TYPE ST_ECB :
STRUCT
	Status AT %I* : BOOL;
	Reset AT %Q* : BOOL;
	Name : STRING;
	Description : STRING;
END_STRUCT
END_TYPE

(* stored: Version 1.1.0.1, ProductVersion 3.1.4026.18
   DUT ST_ECB: Id {42e0f514-4cda-48f0-a408-87660953d3ed} *)
